TYPE ST_SafetyDescription :
STRUCT
	sSafetyName : STRING(nMAX_SAFETY_NAME);
	eSafetyType : E_SafetyType;
	sLocation  : STRING(nMAX_LOCATION_NAME);
END_STRUCT
END_TYPE

(* stored: Version 1.1.0.1, ProductVersion 3.1.4024.11
   DUT ST_SafetyDescription: Id {6dea37be-1adc-41e4-9cc9-dc56187ec785} *)
